SUBAPPLICATION Uebung_034b_AUDI (* LONG_PRESS_HOLD-Eingang auf PWM Ausgang (Adapter Version) mit Terminal-Ausgabe *)
  (* Standard: 61499-2; Description: Copyright (c) 2023 Meisterschulen am Ostbahnhof This program and the accompanying materials are made available under the terms of the Eclipse Public License 2.0 which is available at https://www.eclipse.org/legal/epl-2.0/ SPDX-License-Identifier: EPL-2.0 *)
  (* Version 1.1, 2026-04-21, Franz Höpfinger, Meisterschulen am Ostbahnhof, Added terminal output for counter value *)
  (* Version 1.0, 2023-10-23, Franz Höpfinger, Meisterschulen am Ostbahnhof, initial API and implementation and/or initial documentation *)
  PACKAGE Uebungen;
  IMPORT Uebungen::const::UT::DefaultPool::OutputNumber_N1;
  IMPORT logiBUS::io::DI::logiBUS_DI::Input_I1;
  IMPORT logiBUS::io::DI::logiBUS_DI::Input_I2;
  IMPORT logiBUS::io::DI::logiBUS_DI::Input_I3;
  IMPORT logiBUS::io::DI::logiBUS_DI::Input_I4;
  IMPORT logiBUS::io::DI::logiBUS_DI_Events::BUTTON_LONG_PRESS_HOLD;
  IMPORT logiBUS::io::DI::logiBUS_DI_Events::BUTTON_SINGLE_CLICK;
  IMPORT logiBUS::io::DQ::logiBUS_DO::Output_Q1;
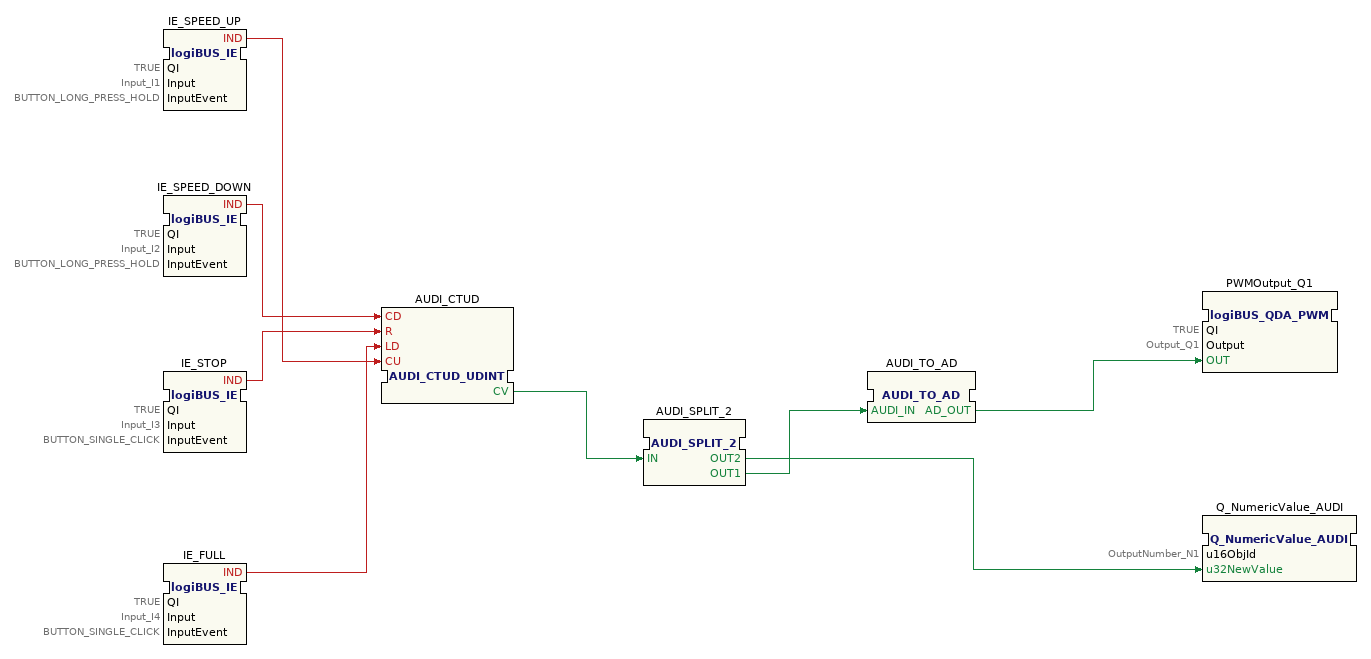
  FBS
    PWMOutput_Q1 : logiBUS::io::DQ::logiBUS_QDA_PWM(QI := TRUE, Output := Output_Q1);
    IE_SPEED_UP : logiBUS::io::DI::logiBUS_IE(QI := TRUE, Input := Input_I1, InputEvent := BUTTON_LONG_PRESS_HOLD);
    IE_SPEED_DOWN : logiBUS::io::DI::logiBUS_IE(QI := TRUE, Input := Input_I2, InputEvent := BUTTON_LONG_PRESS_HOLD);
    IE_STOP : logiBUS::io::DI::logiBUS_IE(QI := TRUE, Input := Input_I3, InputEvent := BUTTON_SINGLE_CLICK);
    IE_FULL : logiBUS::io::DI::logiBUS_IE(QI := TRUE, Input := Input_I4, InputEvent := BUTTON_SINGLE_CLICK);
    AUDI_CTUD : adapter::events::unidirectional::AUDI_CTUD_UDINT;
    Q_NumericValue_AUDI : isobus::UT::Q::Q_NumericValue_AUDI(u16ObjId := OutputNumber_N1);
    AUDI_SPLIT_2 : adapter::events::unidirectional::AUDI_SPLIT_2;
    AUDI_TO_AD : adapter::conversion::unidirectional::AUDI_TO_AD;
  END_FBS
  EVENT_CONNECTIONS
    IE_SPEED_DOWN.IND TO AUDI_CTUD.CD;
    IE_STOP.IND TO AUDI_CTUD.R;
    IE_FULL.IND TO AUDI_CTUD.LD;
    IE_SPEED_UP.IND TO AUDI_CTUD.CU;
  END_CONNECTIONS
  ADAPTER_CONNECTIONS
    AUDI_CTUD.CV TO AUDI_SPLIT_2.IN;
    AUDI_SPLIT_2.OUT2 TO Q_NumericValue_AUDI.u32NewValue;
    AUDI_SPLIT_2.OUT1 TO AUDI_TO_AD.AUDI_IN;
    AUDI_TO_AD.AD_OUT TO PWMOutput_Q1.OUT;
  END_CONNECTIONS
END_SUBAPPLICATION
